// TIA Portal V20 export
TYPE "typeFDoorElement"
// stored: Access Published, IsFailsafeCompliant true, Namespace Safety
   STRUCT
      FDoor1 : Bool;   // EC Top Gate
      FDoor2 : Bool;   // EC LH Gate
      FDoor3 : Bool;   // EC RH Gate
      FDoor4 : Bool;   // Cutter Gate
      FDoor5 : Bool;   // Magazine system Gate
      FDoor6 : Bool;   // Conveyor Area Gate
      FDoor7 : Bool;   // Central Aisle Gate
      FDoor8 : Bool;   // Stack30 Cover Gate
      FDoor9 : Bool;   // Stack40 Cover Gate
   END_STRUCT;
END_TYPE
